{attribute 'TcGenerated'}
// This function has been automatically generated from the project information.
VAR_GLOBAL CONSTANT
	{attribute 'const_non_replaced'}
	{attribute 'linkalways'}
	stLibVersion_lcls2-cc-lib : ST_LibVersion := (iMajor := 1, iMinor := 0, iBuild := 1, iRevision := 0, sVersion := '1.0.1');
END_VAR

(* stored: Version 1.1.0.1, ProductVersion 3.1.4022.18
   GVL Global_Version: Id 36eb4cb5-ac55-4c33-b0b3-c15795ab30a8 *)
